// TIA Portal V15.1 export
// export: Created 2026-01-15T16:29:41.5964636Z, ExportSetting WithDefaults, WithReadOnly, DisplayName Totally Integrated Automation Portal, DisplayVersion V15.1 Update 8, DisplayName TIA Portal Openness, DisplayVersion V15.1 Update 8, DisplayName STEP 7 Professional, DisplayVersion V15.1 Update 8, DisplayName WinCC Advanced, DisplayVersion V15.1 Update 8
FUNCTION "3.OUTPUT_PLC" : Void   // FC3, LAD
{ S7_Optimized_Access := 'TRUE' }
VERSION : 0.1
// stored: AutoNumber false, CodeModifiedDate 2025-08-27T17:07:28.4518091Z, CompileDate 2026-01-15T16:25:55.7493553Z, CreationDate 2026-01-15T16:22:49.8270549Z, HandleErrorsWithinBlock false, InterfaceModifiedDate 2022-06-07T03:40:45.7898546Z, IsConsistent true, IsIECCheckEnabled false, IsKnowHowProtected false, IsWriteProtected false, LibraryConformanceStatus The object is library-conformant., ModifiedDate 2025-08-27T17:07:28.4518091Z, ParameterModified 2022-06-07T03:40:45.7898546Z, PLCSimAdvancedSupport false, SetENOAutomatically False, StructureModified 2022-06-07T03:40:45.7898546Z, UDAEnableTagReadback false
   VAR_INPUT
      A1 : Bool;
      M1 : Bool;
      A2 : Bool;
      M2 : Bool;
      A3 : Bool;
      M3 : Bool;
      A4 : Bool;
      M4 : Bool;
   END_VAR
   VAR_OUTPUT
      OUT1 : Bool;
      OUT2 : Bool;
      OUT3 : Bool;
      OUT4 : Bool;
   END_VAR
BEGIN

REGION Network 1
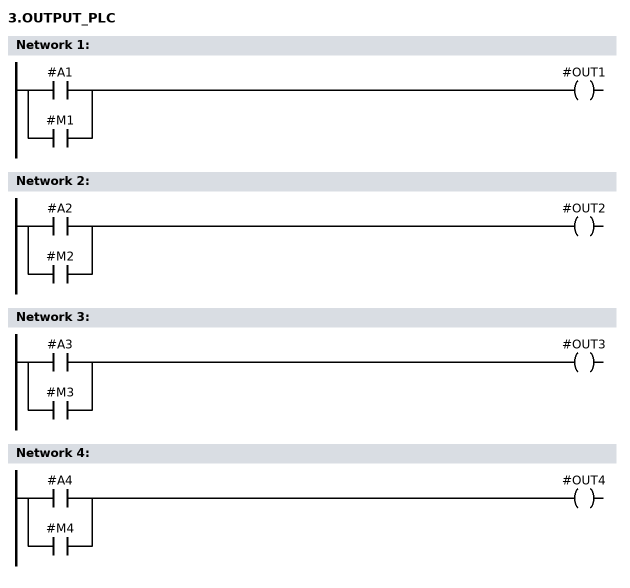
   RUNG wire#powerrail
      Contact( #A1 )
      wire#w1
      Coil( #OUT1 )
   END_RUNG
   RUNG wire#powerrail
      Contact( #M1 )
   END_RUNG wire#w1
   // the same network as SCL:
   #OUT1 := #A1 OR #M1;
END_REGION

REGION Network 2
   RUNG wire#powerrail
      Contact( #A2 )
      wire#w1
      Coil( #OUT2 )
   END_RUNG
   RUNG wire#powerrail
      Contact( #M2 )
   END_RUNG wire#w1
   // the same network as SCL:
   #OUT2 := #A2 OR #M2;
END_REGION

REGION Network 3
   RUNG wire#powerrail
      Contact( #A3 )
      wire#w1
      Coil( #OUT3 )
   END_RUNG
   RUNG wire#powerrail
      Contact( #M3 )
   END_RUNG wire#w1
   // the same network as SCL:
   #OUT3 := #A3 OR #M3;
END_REGION

REGION Network 4
   RUNG wire#powerrail
      Contact( #A4 )
      wire#w1
      Coil( #OUT4 )
   END_RUNG
   RUNG wire#powerrail
      Contact( #M4 )
   END_RUNG wire#w1
   // the same network as SCL:
   #OUT4 := #A4 OR #M4;
END_REGION
END_FUNCTION
